PROGRAM TestTorqueProfile
VAR
TorCmdMax : DINT := TRUNC( 3.0 * 1E6 / 10000);// TC*10e6/0x6076
MyTime : INT :=0;
tTimerValue     : LTIME ;//:= T#0S;
tTimeHr : UDINT;
END_VAR


//IF ServoCtrl.TargetTorque > TorCmdMax THEN
//	Ds402.DirUp := FALSE;
//END_IF
//
//IF ServoCtrl.TargetTorque < -TorCmdMax THEN
//	Ds402.DirUp := TRUE;
//END_IF
//		
//IF Ds402.DirUp THEN 
//	ServoCtrl.TargetTorque := ServoCtrl.TargetTorque+1;
//ELSE
//	ServoCtrl.TargetTorque := ServoCtrl.TargetTorque-1;
//END_IF

tTimerValue := LTIME();
tTimeHr := LTIME_TO_UDINT(tTimerValue) MOD  67108864 ;// 

MyTime := (MyTime +1) MOD  2048 ;
//for Ts=100usec: ServoCtrl.TargetTorque := TRUNC_INT( TorCmdMax * SIN(  tTimeHr * 6.28 *32.0 / 67108864.0 ));

// for Ts = 1ms
ServoCtrl.TargetTorque := TRUNC_INT( TorCmdMax * SIN(  tTimeHr * 6.28 *4.0 / 67108864.0 ));

// ServoCtrl.TargetTorque := TRUNC_INT( TorCmdMax * SIN(  MyTime * 6.28 * 25  / 2048.0 ));

END_PROGRAM

(* stored: Version 1.1.0.1, ProductVersion 3.1.4024.6
   POU TestTorqueProfile: Id {3f6cf7d5-b6f9-460f-bfd8-22f60a81aa8e}, SpecialFunc None *)
